// TIA Portal V20 export
VAR_GLOBAL   // PLC tag table "ASi"
   "ASiGW-MCC100-bw23-C1: Input" AT %I2300.0 : "tASiGW-MCC100-bw23-C1: Input";
   "ASiGW-MCC100-bw23-C1: Output" AT %Q2300.0 : "tASiGW-MCC100-bw23-C1: Output";
   "ASiGW-MCC100-bw23-C1: ConfigErr" AT %I2364.0 : "Config/PeriErr";
   "ASiGW-MCC100-bw23-C1: PeriErr" AT %I2372.0 : "Config/PeriErr";
END_VAR
